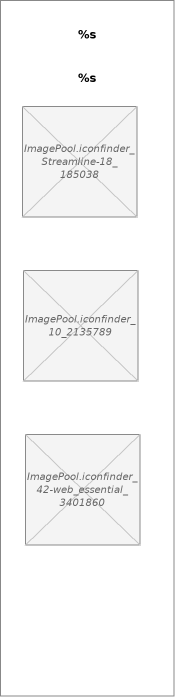
VISUALIZATION VISU_FRAME  // 175x697
VAR_INPUT
	
sDayTime : STRING;
sTime : STRING;

END_VAR
    Rectangle (0,0 175x697)
    Image (23,270 115x111), image: ImagePool.iconfinder_10_2135789
        OnMouseClick: change screen: Visualization_2
    Rectangle (23,385 117x33), text list: 'TextList', text index: 1
    Image (22,106 115x111), image: ImagePool.iconfinder_Streamline-18_185038
        OnMouseClick: change screen: Visualization_3
    Rectangle (22,222 117x33), text list: 'TextList', text index: 2
    Image (25,434 115x111), image: ImagePool.iconfinder_42-web_essential_3401860
        OnMouseClick: change screen: Visualization_1
    Rectangle (25,550 117x33), text list: 'TextList', text index: 0
    Rectangle (12,17 151x35), "%s", text variable: sDayTime
    Rectangle (12,61 151x34), "%s", text variable: sTime
END_VISUALIZATION

(* stored: Version 1.1.0.1, ProductVersion 3.1.4024.4
   Visu VISU_FRAME: Id {9748bc20-9944-4876-a566-f8d280a556b8} *)
